PROGRAM INTERNAL PRG_TEST
VAR
	// ManualControl
	bInitDone : BOOL;
	fbFaultHandler 			: Fb_FaultHandler; 
	fbDevValve 				: FB_DevValve;
END_VAR


// Parameters
	// NOTE: fbParameterHandler should contain the parameters of fbDevValve. 
	// Parameter values are persistent

	IF NOT bInitDone THEN
		bInitDone := TRUE;
		fbDevValve.Init(
			nId := 1,
			nParentId := 0,
			eResetState := E_ValveResetState.Res_Idle,
			eSafeState := E_ValveResetState.Res_Idle
		);
	END_IF
	
	fbFaultHandler();
	fbDevValve(
		refFbFault := fbFaultHandler,
		refFbManualCtrl	:= GVL_DevManual.fbManualControler,
	);

	GVL_Parameters.fbParameterHandler();

GVL_HMI.fbHMIControl();

END_PROGRAM

(* stored: Version 1.1.0.1, ProductVersion 3.1.4024.11
   POU PRG_TEST: Id {b132eb66-7e41-469d-9de4-883897ec1165}, SpecialFunc None *)
